PROGRAM MAIN
VAR
END_VAR

P_EIB_KNX();

END_PROGRAM

(* stored: Version 1.1.0.1, ProductVersion 3.1.4022.18
   POU MAIN: Id {0ca77731-1f37-418e-a16b-3f688071b11d}, SpecialFunc None *)
